Staubli VAL3: calculation.pgx

program calculation(num x_nX1, num x_nX2, num x_nX3, num x_nX4, num x_nY1, num x_nY2, num x_nY3, num x_nY4, num x_nZ1, num x_nZ2, num x_nZ3, num x_nZ4)
  local num l_nTemp
  local num l_nI
  local num l_nGesamtX
  local num l_nGesamtY
  local num l_nGesamtZ
begin
  //-----------------------------------------------------------------------
  //Header begin
  //Description of program
  //  This program calculates the tool to find the X, Y, Z components
  //
  //Input parameters
  //  num x_nX1 to x_nX4
  //  num x_nY1 to x_nY4
  //  num x_nZ1 to x_nZ4
  //
  //Traceability
  //  Creation : 07-04-08 - f.Rob
  //  Used without modification for SLAC  KN  17aug2009
  //Header end
  //-----------------------------------------------------------------------

  nScX=x_nY1*x_nX3*x_nX3*x_nZ2+x_nX1*x_nX1*x_nY2*x_nZ3-x_nX1*x_nX1*x_nY3*x_nZ2-x_nX2*x_nX2*x_nY1*x_nZ3
  nScX=nScX-x_nX3*x_nX3*x_nY2*x_nZ1-x_nY1*x_nY2*x_nY2*x_nZ3-x_nY1*x_nX4*x_nX4*x_nZ2+x_nY1*x_nY3*x_nY3*x_nZ2
  nScX=nScX+x_nY2*x_nZ1*x_nX4*x_nX4-x_nY2*x_nZ1*x_nY3*x_nY3-x_nX1*x_nX1*x_nY2*x_nZ4+x_nX1*x_nX1*x_nZ2*x_nY4
  nScX=nScX+x_nX2*x_nX2*x_nY1*x_nZ4-x_nX2*x_nX2*x_nZ1*x_nY4+x_nY1*x_nY1*x_nY2*x_nZ3-x_nY1*x_nY1*x_nY3*x_nZ2
  nScX=nScX+x_nY2*x_nY2*x_nZ1*x_nY3-x_nY1*x_nZ2*x_nY4*x_nY4+x_nY1*x_nZ2*x_nZ3*x_nZ3-x_nY1*x_nX3*x_nX3*x_nZ4
  nScX=nScX+x_nY1*x_nY2*x_nY2*x_nZ4+x_nY1*x_nX4*x_nX4*x_nZ3-x_nY1*x_nZ2*x_nZ2*x_nZ3+x_nY2*x_nZ1*x_nY4*x_nY4
  nScX=nScX-x_nY2*x_nZ1*x_nZ3*x_nZ3+x_nY2*x_nZ1*x_nZ1*x_nZ3+x_nZ1*x_nY3*x_nZ2*x_nZ2-x_nZ1*x_nX4*x_nX4*x_nY3
  nScX=nScX+x_nX1*x_nX1*x_nY3*x_nZ4-x_nX1*x_nX1*x_nY4*x_nZ3-x_nY1*x_nY1*x_nY2*x_nZ4+x_nY1*x_nY1*x_nZ2*x_nY4
  nScX=nScX+x_nX3*x_nX3*x_nZ1*x_nY4-x_nY2*x_nY2*x_nZ1*x_nY4-x_nZ1*x_nZ1*x_nY3*x_nZ2-x_nY1*x_nZ2*x_nZ4*x_nZ4
  nScX=nScX-x_nY1*x_nY3*x_nY3*x_nZ4+x_nY1*x_nZ2*x_nZ2*x_nZ4+x_nY1*x_nY4*x_nY4*x_nZ3+x_nY2*x_nZ1*x_nZ4*x_nZ4
  nScX=nScX-x_nY2*x_nZ1*x_nZ1*x_nZ4-x_nY2*x_nX4*x_nX4*x_nZ3-x_nZ1*x_nY3*x_nY4*x_nY4+x_nZ1*x_nY3*x_nY3*x_nY4
  nScX=nScX-x_nZ1*x_nZ2*x_nZ2*x_nY4-x_nX2*x_nX2*x_nY3*x_nZ4+x_nX2*x_nX2*x_nY4*x_nZ3+x_nY1*x_nY1*x_nY3*x_nZ4
  nScX=nScX-x_nY1*x_nY1*x_nY4*x_nZ3+x_nX3*x_nX3*x_nY2*x_nZ4-x_nX3*x_nX3*x_nZ2*x_nY4+x_nZ1*x_nZ1*x_nZ2*x_nY4
  nScX=nScX+x_nX4*x_nX4*x_nY3*x_nZ2+x_nY1*x_nZ3*x_nZ4*x_nZ4-x_nY1*x_nZ3*x_nZ3*x_nZ4+x_nY2*x_nY3*x_nY3*x_nZ4
  nScX=nScX-x_nY2*x_nY4*x_nY4*x_nZ3-x_nZ1*x_nY3*x_nZ4*x_nZ4+x_nZ1*x_nY4*x_nZ3*x_nZ3+x_nY3*x_nZ2*x_nY4*x_nY4
  nScX=nScX-x_nY2*x_nY2*x_nY3*x_nZ4+x_nY2*x_nY2*x_nY4*x_nZ3+x_nZ1*x_nZ1*x_nY3*x_nZ4-x_nZ1*x_nZ1*x_nY4*x_nZ3
  nScX=nScX-x_nY3*x_nY3*x_nZ2*x_nY4-x_nY2*x_nZ3*x_nZ4*x_nZ4+x_nY2*x_nZ3*x_nZ3*x_nZ4+x_nY3*x_nZ2*x_nZ4*x_nZ4
  nScX=nScX-x_nY3*x_nZ2*x_nZ2*x_nZ4-x_nZ2*x_nY4*x_nZ3*x_nZ3+x_nZ2*x_nZ2*x_nY4*x_nZ3+x_nX2*x_nX2*x_nZ1*x_nY3
  l_nTemp=2*x_nX1*x_nY2*x_nZ3-2*x_nX1*x_nY3*x_nZ2-2*x_nX2*x_nY1*x_nZ3+2*x_nX2*x_nZ1*x_nY3+2*x_nY1*x_nX3*x_nZ2
  l_nTemp=l_nTemp-2*x_nX3*x_nY2*x_nZ1-2*x_nX1*x_nY2*x_nZ4+2*x_nX1*x_nZ2*x_nY4+2*x_nX2*x_nY1*x_nZ4-2*x_nX2*x_nZ1*x_nY4-2*x_nY1*x_nX4*x_nZ2
  l_nTemp=l_nTemp+2*x_nY2*x_nZ1*x_nX4+2*x_nX1*x_nY3*x_nZ4-2*x_nX1*x_nY4*x_nZ3-2*x_nY1*x_nX3*x_nZ4+2*x_nY1*x_nX4*x_nZ3+2*x_nX3*x_nZ1*x_nY4
  l_nTemp=l_nTemp-2*x_nZ1*x_nX4*x_nY3-2*x_nX2*x_nY3*x_nZ4+2*x_nX2*x_nY4*x_nZ3+2*x_nX3*x_nY2*x_nZ4-2*x_nX3*x_nZ2*x_nY4-2*x_nY2*x_nX4*x_nZ3
  l_nTemp=l_nTemp+2*x_nX4*x_nY3*x_nZ2
  if abs(l_nTemp)<0.001
    nScX=9999.9999
  else
    nScX=nScX/l_nTemp
  endIf
  nScY=x_nX1*x_nX2*x_nX2*x_nZ3-x_nX1*x_nX3*x_nX3*x_nZ2+x_nX2*x_nX3*x_nX3*x_nZ1-x_nX1*x_nX1*x_nX2*x_nZ3
  nScY=nScY+x_nX1*x_nX1*x_nX3*x_nZ2-x_nX2*x_nX2*x_nX3*x_nZ1-x_nX1*x_nX2*x_nX2*x_nZ4+x_nX1*x_nY2*x_nY2*x_nZ3
  nScY=nScY+x_nX1*x_nX4*x_nX4*x_nZ2-x_nX1*x_nY3*x_nY3*x_nZ2-x_nX2*x_nZ1*x_nX4*x_nX4+x_nX2*x_nZ1*x_nY3*x_nY3
  nScY=nScY-x_nX2*x_nY1*x_nY1*x_nZ3-x_nX3*x_nY2*x_nY2*x_nZ1+x_nX1*x_nX1*x_nX2*x_nZ4-x_nX1*x_nX1*x_nX4*x_nZ2
  nScY=nScY+x_nX2*x_nX2*x_nZ1*x_nX4+x_nY1*x_nY1*x_nX3*x_nZ2+x_nX1*x_nZ2*x_nY4*x_nY4-x_nX1*x_nZ2*x_nZ3*x_nZ3
  nScY=nScY+x_nX1*x_nX3*x_nX3*x_nZ4-x_nX1*x_nY2*x_nY2*x_nZ4-x_nX1*x_nX4*x_nX4*x_nZ3+x_nX1*x_nZ2*x_nZ2*x_nZ3
  nScY=nScY-x_nX2*x_nZ1*x_nY4*x_nY4+x_nX2*x_nZ1*x_nZ3*x_nZ3+x_nX2*x_nY1*x_nY1*x_nZ4-x_nX2*x_nZ1*x_nZ1*x_nZ3
  nScY=nScY+x_nX3*x_nZ1*x_nX4*x_nX4-x_nX3*x_nZ1*x_nZ2*x_nZ2+x_nX3*x_nZ1*x_nZ1*x_nZ2-x_nX1*x_nX1*x_nX3*x_nZ4
  nScY=nScY+x_nX1*x_nX1*x_nX4*x_nZ3-x_nY1*x_nY1*x_nX4*x_nZ2-x_nX3*x_nX3*x_nZ1*x_nX4+x_nY2*x_nY2*x_nZ1*x_nX4
  nScY=nScY+x_nX1*x_nZ2*x_nZ4*x_nZ4+x_nX1*x_nY3*x_nY3*x_nZ4-x_nX1*x_nZ2*x_nZ2*x_nZ4-x_nX1*x_nY4*x_nY4*x_nZ3
  nScY=nScY-x_nX2*x_nZ1*x_nZ4*x_nZ4-x_nX2*x_nX3*x_nX3*x_nZ4+x_nX2*x_nZ1*x_nZ1*x_nZ4+x_nX2*x_nX4*x_nX4*x_nZ3
  nScY=nScY+x_nX3*x_nZ1*x_nY4*x_nY4-x_nX3*x_nX4*x_nX4*x_nZ2-x_nZ1*x_nX4*x_nY3*x_nY3+x_nZ1*x_nX4*x_nZ2*x_nZ2
  nScY=nScY+x_nX2*x_nX2*x_nX3*x_nZ4-x_nX2*x_nX2*x_nX4*x_nZ3-x_nY1*x_nY1*x_nX3*x_nZ4+x_nY1*x_nY1*x_nX4*x_nZ3
  nScY=nScY+x_nX3*x_nX3*x_nX4*x_nZ2-x_nZ1*x_nZ1*x_nX4*x_nZ2-x_nX1*x_nZ3*x_nZ4*x_nZ4+x_nX1*x_nZ3*x_nZ3*x_nZ4
  nScY=nScY-x_nX2*x_nY3*x_nY3*x_nZ4+x_nX2*x_nY4*x_nY4*x_nZ3+x_nX3*x_nZ1*x_nZ4*x_nZ4-x_nX3*x_nZ2*x_nY4*x_nY4
  nScY=nScY+x_nX3*x_nY2*x_nY2*x_nZ4-x_nX3*x_nZ1*x_nZ1*x_nZ4-x_nZ1*x_nX4*x_nZ3*x_nZ3+x_nX4*x_nY3*x_nY3*x_nZ2
  nScY=nScY-x_nY2*x_nY2*x_nX4*x_nZ3+x_nZ1*x_nZ1*x_nX4*x_nZ3+x_nX2*x_nZ3*x_nZ4*x_nZ4-x_nX2*x_nZ3*x_nZ3*x_nZ4
  nScY=nScY-x_nX3*x_nZ2*x_nZ4*x_nZ4+x_nX3*x_nZ2*x_nZ2*x_nZ4+x_nX4*x_nZ2*x_nZ3*x_nZ3-x_nX4*x_nZ2*x_nZ2*x_nZ3
  l_nTemp=2*x_nX1*x_nY2*x_nZ3-2*x_nX1*x_nY3*x_nZ2-2*x_nX2*x_nY1*x_nZ3+2*x_nX2*x_nZ1*x_nY3
  l_nTemp=l_nTemp+2*x_nY1*x_nX3*x_nZ2-2*x_nX3*x_nY2*x_nZ1-2*x_nX1*x_nY2*x_nZ4+2*x_nX1*x_nZ2*x_nY4+2*x_nX2*x_nY1*x_nZ4-2*x_nX2*x_nZ1*x_nY4
  l_nTemp=l_nTemp-2*x_nY1*x_nX4*x_nZ2+2*x_nY2*x_nZ1*x_nX4+2*x_nX1*x_nY3*x_nZ4-2*x_nX1*x_nY4*x_nZ3-2*x_nY1*x_nX3*x_nZ4+2*x_nY1*x_nX4*x_nZ3
  l_nTemp=l_nTemp+2*x_nX3*x_nZ1*x_nY4-2*x_nZ1*x_nX4*x_nY3-2*x_nX2*x_nY3*x_nZ4+2*x_nX2*x_nY4*x_nZ3+2*x_nX3*x_nY2*x_nZ4-2*x_nX3*x_nZ2*x_nY4
  l_nTemp=l_nTemp-2*x_nY2*x_nX4*x_nZ3+2*x_nX4*x_nY3*x_nZ2
  if abs(l_nTemp)<0.001
    nScY=9999.9999
  else
    nScY=nScY/l_nTemp
  endIf
  nScZ=x_nX1*x_nX3*x_nX3*x_nY2-x_nX1*x_nX2*x_nX2*x_nY3-x_nX2*x_nY1*x_nX3*x_nX3+x_nX1*x_nX1*x_nX2*x_nY3
  nScZ=nScZ-x_nX1*x_nX1*x_nX3*x_nY2+x_nX2*x_nX2*x_nY1*x_nX3-x_nX1*x_nY2*x_nX4*x_nX4+x_nX1*x_nY2*x_nY3*x_nY3
  nScZ=nScZ+x_nX1*x_nX2*x_nX2*x_nY4-x_nX1*x_nY2*x_nY2*x_nY3+x_nX2*x_nY1*x_nX4*x_nX4-x_nX2*x_nY1*x_nY3*x_nY3
  nScZ=nScZ+x_nX2*x_nY1*x_nY1*x_nY3+x_nY1*x_nX3*x_nY2*x_nY2-x_nX1*x_nX1*x_nX2*x_nY4+x_nX1*x_nX1*x_nY2*x_nX4
  nScZ=nScZ-x_nX2*x_nX2*x_nY1*x_nX4-x_nY1*x_nY1*x_nX3*x_nY2-x_nX1*x_nY2*x_nY4*x_nY4+x_nX1*x_nY2*x_nZ3*x_nZ3
  nScZ=nScZ-x_nX1*x_nY3*x_nZ2*x_nZ2-x_nX1*x_nX3*x_nX3*x_nY4+x_nX1*x_nY2*x_nY2*x_nY4+x_nX1*x_nX4*x_nX4*x_nY3
  nScZ=nScZ+x_nX2*x_nY1*x_nY4*x_nY4-x_nX2*x_nY1*x_nZ3*x_nZ3-x_nX2*x_nY1*x_nY1*x_nY4+x_nX2*x_nZ1*x_nZ1*x_nY3
  nScZ=nScZ-x_nY1*x_nX3*x_nX4*x_nX4+x_nY1*x_nX3*x_nZ2*x_nZ2+x_nY1*x_nX3*x_nX3*x_nX4-x_nY1*x_nY2*x_nY2*x_nX4
  nScZ=nScZ-x_nX3*x_nY2*x_nZ1*x_nZ1+x_nX1*x_nX1*x_nX3*x_nY4-x_nX1*x_nX1*x_nX4*x_nY3+x_nY1*x_nY1*x_nY2*x_nX4
  nScZ=nScZ-x_nX1*x_nY2*x_nZ4*x_nZ4+x_nX1*x_nY3*x_nY4*x_nY4-x_nX1*x_nY3*x_nY3*x_nY4+x_nX1*x_nZ2*x_nZ2*x_nY4
  nScZ=nScZ+x_nX2*x_nY1*x_nZ4*x_nZ4+x_nX2*x_nX3*x_nX3*x_nY4-x_nX2*x_nZ1*x_nZ1*x_nY4-x_nX2*x_nX4*x_nX4*x_nY3
  nScZ=nScZ-x_nY1*x_nX3*x_nY4*x_nY4+x_nY1*x_nX4*x_nY3*x_nY3-x_nY1*x_nX4*x_nZ2*x_nZ2+x_nX3*x_nY2*x_nX4*x_nX4
  nScZ=nScZ+x_nY2*x_nZ1*x_nZ1*x_nX4-x_nX2*x_nX2*x_nX3*x_nY4+x_nX2*x_nX2*x_nX4*x_nY3+x_nY1*x_nY1*x_nX3*x_nY4
  nScZ=nScZ-x_nY1*x_nY1*x_nX4*x_nY3-x_nX3*x_nX3*x_nY2*x_nX4+x_nX1*x_nY3*x_nZ4*x_nZ4-x_nX1*x_nY4*x_nZ3*x_nZ3
  nScZ=nScZ-x_nX2*x_nY3*x_nY4*x_nY4+x_nX2*x_nY3*x_nY3*x_nY4-x_nY1*x_nX3*x_nZ4*x_nZ4+x_nY1*x_nX4*x_nZ3*x_nZ3
  nScZ=nScZ+x_nX3*x_nY2*x_nY4*x_nY4-x_nX3*x_nY2*x_nY2*x_nY4+x_nX3*x_nZ1*x_nZ1*x_nY4-x_nY2*x_nX4*x_nY3*x_nY3
  nScZ=nScZ+x_nY2*x_nY2*x_nX4*x_nY3-x_nZ1*x_nZ1*x_nX4*x_nY3-x_nX2*x_nY3*x_nZ4*x_nZ4+x_nX2*x_nY4*x_nZ3*x_nZ3
  nScZ=nScZ+x_nX3*x_nY2*x_nZ4*x_nZ4-x_nX3*x_nZ2*x_nZ2*x_nY4-x_nY2*x_nX4*x_nZ3*x_nZ3+x_nX4*x_nY3*x_nZ2*x_nZ2
  l_nTemp=2*x_nX1*x_nY2*x_nZ3-2*x_nX1*x_nY3*x_nZ2-2*x_nX2*x_nY1*x_nZ3+2*x_nX2*x_nZ1*x_nY3+2*x_nY1*x_nX3*x_nZ2-2*x_nX3*x_nY2*x_nZ1
  l_nTemp=l_nTemp-2*x_nX1*x_nY2*x_nZ4+2*x_nX1*x_nZ2*x_nY4+2*x_nX2*x_nY1*x_nZ4-2*x_nX2*x_nZ1*x_nY4-2*x_nY1*x_nX4*x_nZ2+2*x_nY2*x_nZ1*x_nX4
  l_nTemp=l_nTemp+2*x_nX1*x_nY3*x_nZ4-2*x_nX1*x_nY4*x_nZ3-2*x_nY1*x_nX3*x_nZ4+2*x_nY1*x_nX4*x_nZ3+2*x_nX3*x_nZ1*x_nY4-2*x_nZ1*x_nX4*x_nY3
  l_nTemp=l_nTemp-2*x_nX2*x_nY3*x_nZ4+2*x_nX2*x_nY4*x_nZ3+2*x_nX3*x_nY2*x_nZ4-2*x_nX3*x_nZ2*x_nY4-2*x_nY2*x_nX4*x_nZ3+2*x_nX4*x_nY3*x_nZ2
  if abs(l_nTemp)<0.001
    nScZ=9999.9999
  else
    nScZ=nScZ/l_nTemp
  endIf
  if ((nScX==9999.9999) or (nScY==9999.9999) or (nScZ==9999.9999))
    bAbort=true
    call valSetBack()
  else
    bAbort=false
    //Theoretical Center of Sphere
    trCenter={nScX,nScY,nScZ,0,0,0}
    //Inverse sphere * center
    for l_nI=0 to 3
      trTempTool[l_nI]=!trSphere[l_nI]*trCenter
    endFor
    l_nGesamtX=0
    l_nGesamtY=0
    l_nGesamtZ=0
    for l_nI=0 to 3
      l_nGesamtX=l_nGesamtX+trTempTool[l_nI].x
      l_nGesamtY=l_nGesamtY+trTempTool[l_nI].y
      l_nGesamtZ=l_nGesamtZ+trTempTool[l_nI].z
    endFor
    nToolX=l_nGesamtX/4
    nToolY=l_nGesamtY/4
    nToolZ=l_nGesamtZ/4
  endIf
end
